Universal Robots PolyScope program: TEST_SUB_106B.urp

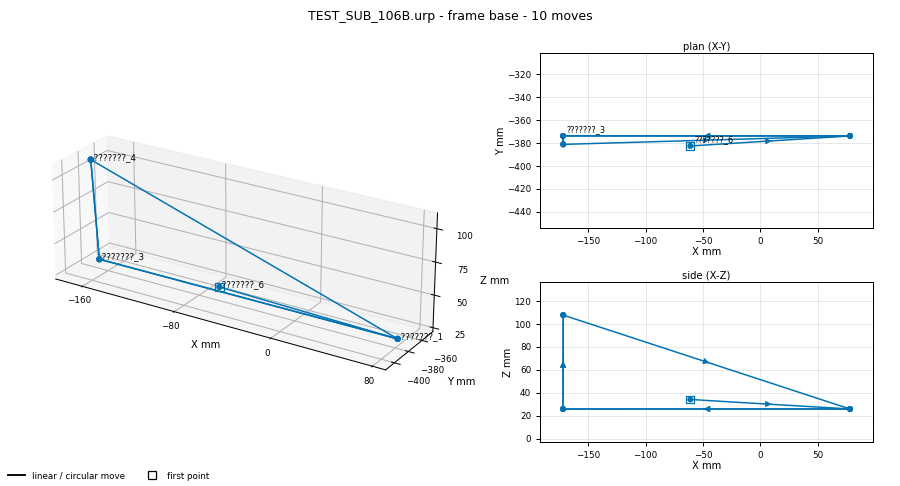
[picture p0: tool path of TEST_SUB_106B.urp in frame base, 10 of 10 moves have a stored position in this frame; points joined in program order, loops and branches not executed]
Program TEST_SUB_106B (installation=GD directory=/programs/GD createdIn=5.13.0 lastSavedIn=5.13.0 robotSerialNumber=20205000017)
Calibrated DH parameters: a=[-0.000157, -0.56303, -0.236706, -0.000074, -0.000109, 0]; d=[0.181705, 47.632387, 369.599619, -417.058513, 0.119878, 0.115667]; alpha=[1.570881, -0.005074, -0.001247, 1.56886, -1.570997, 0]; deltaTheta=[0, -0.405485, 5.544791, 1.143886, -0.000009, -0.000001]
InitVariablesNode
BeforeStart
  Script file /home/ros/ursim-5.13.0.113898/programs/GD/CONTROL/ALIGN_AXIS.script
    | def GET_NORM_VEC(p,axis=2):
    |   rot=p[0.0, 0.0, 0.0, p[3], p[4], p[5]]
    |   vec=p[0.0, 0.0, 0.0, 0.0, 0.0, 0.0]
    |   vec[axis]=1.0
    |   norm_p=pose_trans(rot,vec)
    |   return [norm_p[0], norm_p[1], norm_p[2]]
    | end
    | 
    | def GET_INNER_PRODUCT(v1,v2):
    |   return v1[0]*v2[0]+v1[1]*v2[1]+v1[2]*v2[2]
    | end
    | def GET_OUTER_PRODUCT(v1,v2):
    |   x=v1[1]*v2[2]-v1[2]*v2[1]
    |   y=v1[2]*v2[0]-v1[0]*v2[2]
    |   z=v1[0]*v2[1]-v1[1]*v2[0]
    |   return [x,y,z]
    | end
    | def GET_THETA(v1,v2):
    | #  cos=GET_INNER_PRODUCT(v1,v2) / norm(v1) / norm(v2)
    |   cos=GET_INNER_PRODUCT(v1,v2)
    |   g_cos=cos
    |   theta=norm(acos(cos))
    |   return theta
    | end
    | 
    | def GET_ALIGNED_POSE(target,feature,axis=2):
    |   feature_from_target=pose_trans(pose_inv(target),feature)
    |   g_f_from_t=feature_from_target
    |   nz_feature_from_target=GET_NORM_VEC(feature_from_target,axis)
    |   g_nz_f_from_t=nz_feature_from_target
    |   nz_target_from_target=[0.0, 0.0, 0.0]
    |   nz_target_from_target[axis]=1.0
    |   g_nz_t_from_t=nz_target_from_target
    | 
    |   theta=GET_THETA(nz_feature_from_target,nz_target_from_target)
    |   g_theta=theta
    |   rot_vec_n=normalize(GET_OUTER_PRODUCT(nz_target_from_target,nz_feature_from_target))
    | 
    |   if theta>d2r(90.0):
    |     theta=theta-d2r(180.0)
    |   end
    |   rot_vec=rot_vec_n * (theta)
    |   rot_p=p[0.0,0.0,0.0,rot_vec[0],rot_vec[1],rot_vec[2]]
    |   return pose_trans(target,rot_p)
    | end
    | def GET_ALIGNED_TCP(feature,axis=2):
    |   tcp=get_actual_tcp_pose()
    |   return GET_ALIGNED_POSE(tcp,feature,axis)
    | end
  Script file /home/ros/ursim-5.13.0.113898/programs/GD/CONTROL/align_axis_2.script
    | def get_normal_vector(pose, axis=2):
    |  rot = p[0.0, 0.0, 0.0, pose[3], pose[4], pose[5]]
    | 
    |  v = p[0.0, 0.0, 0.0, 0.0, 0.0, 0.0]
    |  if axis==0:
    |   v[0] = 1.0
    |  elif axis==1:
    |   v[1] = 1.0
    |  else:
    |   v[2] = 1.0
    |  end
    | 
    |  normal_p = pose_trans(rot, v)
    |  normal_vector = [normal_p[0], normal_p[1], normal_p[2]]
    |  return normal_vector
    | end
    | 
    | def get_inner_product(v1, v2):
    |  return v1[0]*v2[0] + v1[1]*v2[1] + v1[2]*v2[2]
    | end
    | 
    | def get_theta(v1, v2):
    |  cos = get_inner_product(v1, v2) / norm(v1) / norm(v2)
    |  theta_pn = acos(cos)
    |  theta = norm(theta_pn)
    |  return theta
    | end
    | 
    | def get_outer_product(v1, v2):
    |  x = v1[1]*v2[2] - v1[2]*v2[1]
    |  y = v1[2]*v2[0] - v1[0]*v2[2]
    |  z = v1[0]*v2[1] - v1[1]*v2[0]
    |  return [x,y,z]
    | end
    | 
    | def get_aligned_pose_current_to_base(axis=2):
    |  base = p[0.0, 0.0, 0.0, 0.0, 0.0, 0.0]
    |  pose_cur = get_actual_tcp_pose()
    |  return get_aligned_pose_to_axis(pose_cur, base, axis)
    | end
    | 
    | def get_aligned_pose_current_to_ref(pose_ref, axis=2):
    |  pose_cur = get_actual_tcp_pose()
    |  return get_aligned_pose_to_axis(pose_cur, pose_ref, axis)
    | end
    | 
    | def get_aligned_pose_to_axis(pose_target, pose_ref, axis=2):
    |  pose_ref_from_target = pose_trans(pose_inv(pose_target), pose_ref)
    |  nz_ref_from_target =  get_normal_vector(pose_ref_from_target, axis)
    |  nz_target_from_target = [0.0, 0.0, 1.0]
    | 
    |  if axis == 0:
    |   nz_target_from_target = [1.0, 0.0, 0.0]
    |  elif axis == 1:
    |   nz_target_from_target = [0.0, 1.0, 0.0]
    |  end
    | 
    |  theta = get_theta(nz_ref_from_target, nz_target_from_target)
    |  rot_vector_n = normalize(get_outer_product(nz_target_from_target, nz_ref_from_target))
    | 
    |  if theta > d2r(90.0):
    |   theta = theta - d2r(180.0)
    |  end
    | 
    |  rot_vector = rot_vector_n * (theta)
    | 
    |  pose_rot = p[0.0, 0.0, 0.0, rot_vector[0], rot_vector[1], rot_vector[2]]
    | 
    |  pose_aligned = pose_trans(pose_target, pose_rot)
    | 
    |  return pose_aligned
    | 
    | end
Robot Program (runOnlyOnce=false)
  MoveL speed 250 mm/s, acceleration 50 mm/s^2 (useActiveTCP=false) tcp=TCP_1; feature=Base
    SuppressedNode
      Waypoint ウェイポイント_2: TCP in base x=-24.264 y=-372.872 z=25.863 mm, rx=-0.0592 ry=3.141 rz=-0.0002 rad; joints [-70.474, -66.693, -131.957, -71.332, 89.989, 17.477] deg; TCP offset x=0 y=80 z=420 mm, rx=0 ry=0 rz=0 rad
    SuppressedNode
      Wait Sleep waitTime=0.5
    Waypoint ウェイポイント_6: TCP in base x=-61.068 y=-382.464 z=34.138 mm, rx=0.7542 ry=-2.9409 rz=0.2397 rad; joints [-59.813, -53.273, -138.338, -71.164, 82.262, 0.931] deg
    Wait Sleep waitTime=0.5
  var_5 := p[0.0,0.0,0.0,0.0,0.0,0.0]
  SuppressedNode
    Script: var_5=get_actual_tool_flange_pose()
  SuppressedNode
    Script: var_5[0]=0
  SuppressedNode
    Script: var_5[1]=0
  SuppressedNode
    Script: var_5[0]=0
  Wait Sleep waitTime=0.5
  Set NoAction tcp=TCP_1
  var_4 := GET_ALIGNED_TCP(var_5)
  Wait Sleep waitTime=5
  var_20 := pose_sub(CurrPos,var_4)
  var_21 := pose_trans(pose_inv(CurrPos),var_4)
  Set NoAction tcp=ZERO
  var_1 := get_tcp_offset()
  var_7 := pose_trans(var_1, var_21)
  SuppressedNode
    var_7 := get_aligned_pose_current_to_base()
  SuppressedNode
    MoveL speed 250 mm/s, acceleration 50 mm/s^2 (useActiveTCP=true) feature=Base
      SuppressedNode
        Waypoint ウェイポイント_2: TCP in base x=-24.264 y=-372.872 z=25.863 mm, rx=-0.0592 ry=3.141 rz=-0.0002 rad; joints [-70.474, -66.693, -131.957, -71.332, 89.989, 17.477] deg
      SuppressedNode
        Wait Sleep waitTime=0.5
      Waypoint ウェイポイント_6: TCP in base x=0.269 y=-378.011 z=457.243 mm, rx=0.7542 ry=-2.9409 rz=0.2397 rad; joints [-59.813, -53.273, -138.338, -71.164, 82.262, 0.931] deg
      Wait Sleep waitTime=2
      SuppressedNode
        Waypoint Variable (Variable): variable=var_4
      SuppressedNode
        Wait Sleep waitTime=0.5
  MoveL speed 250 mm/s, acceleration 50 mm/s^2 (useActiveTCP=false) tcp=TCP_1; feature=Base
    Waypoint ウェイポイント_1: TCP in base x=78.379 y=-373.699 z=25.825 mm, rx=-0.2371 ry=3.1325 rz=-0.0004 rad; joints [-56.545, -67.63, -131.248, -71.107, 89.997, 24.798] deg; TCP offset x=0 y=80 z=420 mm, rx=0 ry=0 rz=0 rad
    SuppressedNode
      p1 := CurrPos_p
    Wait Sleep waitTime=1
    SuppressedNode
      p11 := GET_ALIGNED_TCP(p1)
  Script: set_tcp(var_7)
  MoveL speed 250 mm/s, acceleration 50 mm/s^2 (useActiveTCP=true) feature=Base
    Waypoint ウェイポイント_1: TCP in base x=78.379 y=-373.699 z=25.825 mm, rx=-0.2371 ry=3.1325 rz=-0.0004 rad; joints [-56.545, -67.63, -131.248, -71.107, 89.997, 24.798] deg
    Wait Sleep waitTime=1
    SuppressedNode
      Waypoint Variable (Variable): variable=p1
    SuppressedNode
      Wait Sleep waitTime=1
    SuppressedNode
      Waypoint Variable (Variable): variable(name=p11)
    SuppressedNode
      Wait Sleep waitTime=1
    Popup Message (haltProgram=false message=1 done inputType=Text)
  Set NoAction tcp=ZERO
  MoveL speed 250 mm/s, acceleration 50 mm/s^2 (useActiveTCP=false) tcp=TCP_1; feature=Base
    Waypoint ウェイポイント_3: TCP in base x=-172.242 y=-373.664 z=25.794 mm, rx=-0.2375 ry=3.1326 rz=-0.0004 rad; joints [-88.225, -69.95, -129.885, -70.151, 90.002, -6.895] deg
    SuppressedNode
      p2 := CurrPos_p
    Wait Sleep waitTime=1
    SuppressedNode
      p12 := GET_ALIGNED_TCP(p2)
  Script: set_tcp(var_7)
  MoveL speed 250 mm/s, acceleration 50 mm/s^2 (useActiveTCP=true) feature=Base
    Waypoint ウェイポイント_3: TCP in base x=-172.242 y=-373.664 z=25.794 mm, rx=-0.2375 ry=3.1326 rz=-0.0004 rad; joints [-88.225, -69.95, -129.885, -70.151, 90.002, -6.895] deg
    Wait Sleep waitTime=1
    SuppressedNode
      Waypoint Variable (Variable): variable=p2
    SuppressedNode
      Wait Sleep waitTime=1
    SuppressedNode
      Waypoint Variable (Variable): variable(name=p12)
    SuppressedNode
      Wait Sleep waitTime=1
    Popup Message (haltProgram=false message=2 done inputType=Text)
  Set NoAction tcp=ZERO
  MoveL speed 250 mm/s, acceleration 50 mm/s^2 (useActiveTCP=false) tcp=TCP_1; feature=Base
    Waypoint ウェイポイント_4: TCP in base x=-172.007 y=-381.075 z=107.802 mm, rx=-0.2377 ry=3.1326 rz=-0.0003 rad; joints [-88.222, -68.286, -122.359, -79.345, 90.002, -6.902] deg
    SuppressedNode
      p3 := CurrPos_p
    Wait Sleep waitTime=1
    SuppressedNode
      p13 := GET_ALIGNED_TCP(p3)
  Script: set_tcp(var_7)
  MoveL speed 250 mm/s, acceleration 50 mm/s^2 (useActiveTCP=true) feature=Base
    Waypoint ウェイポイント_4: TCP in base x=-172.007 y=-381.075 z=107.802 mm, rx=-0.2377 ry=3.1326 rz=-0.0003 rad; joints [-88.222, -68.286, -122.359, -79.345, 90.002, -6.902] deg
    Wait Sleep waitTime=1
    SuppressedNode
      Waypoint Variable (Variable): variable=p3
    SuppressedNode
      Wait Sleep waitTime=1
    SuppressedNode
      Waypoint Variable (Variable): variable(name=p13)
    SuppressedNode
      Wait Sleep waitTime=1
    Popup Message (haltProgram=false message=3 done inputType=Text)
  Script: CurrPos=get_actual_tool_flange_pose()
  CutOffPos := CurrPos
  var_1 := get_tcp_offset()
  var_2 := pose_trans(CutOffPos,var_1)
  SuppressedNode
    Folder FREE_DRIVE
      Script: freedrive_mode()
      SetPayload (workpieceName=k2)
      Set NoAction tcp=ZERO
      Wait Sleep waitTime=1
      Script: end_freedrive_mode()
      Wait Condition expression=is_steady()
  SetPayload (workpieceName=k10)
  Set NoAction tcp=TCP_1
  Wait Sleep waitTime=0.5
  Folder CUTOFF_POSE
    CutOffPos := CurrPos
    var_6 := CutOffPos
    SuppressedNode
      CutOffPos := p[0.0,0.0,0.0,CutOffPos[3],CutOffPos[4],CutOffPos[5]]
    var_1 := get_tcp_offset()
    var_20 := pose_trans(pose_inv(CutOffPos),var_1)
    SuppressedNode
      CutOffPos := 
    var_4 := p[0.0,0.0,0.0,CutOffPos[3],CutOffPos[4],CutOffPos[5]]
    var_5 := p[0.0,0.0,0.0,0.0,0.0,CutOffPos[5]]
    CutOffPos := pose_trans(var_4,pose_inv(var_5))
    SuppressedNode
      CutOffPos := p[0.0,0.0,0.0,var_5[0],var_5[1],var_5[2]]
    var_20 := pose_trans(pose_inv(CutOffPos),var_1)
    var_21 := pose_trans(var_1,CutOffPos)
    var_2 := pose_trans(CutOffPos,var_1)
  Wait Condition expression=is_steady()
  SuppressedNode
    Script: CurrPos_p=get_actual_tcp_pose()
  SuppressedNode
    CircleMove (OrientationMode=UNCONSTRAINED)
  Script: set_tcp(var_2)
  SuppressedNode
    Folder TRANSFER
      Timer (action=Reset) variable(name=tm_relmove)
      Timer (action=Start) variable=tm_relmove
      ForceStartZ := CurrPos_p[2]
      Force Frame feature=Bucket; selection=[0, 0, 1, 0, 0, 0]; wrench=[0, 0, 40, 0, 0, 0]; limitsForce=[0.01, 0.01, 0.25, 0.174533, 0.174533, 0.174533]; limitsMotion=[0.1, 0.1, 0.1, 0.349066, 0.349066, 0.349066]
        Wait Condition expression=tm_relmove>GPII_TMCutOff or CurrPos_p[2]>ForceStartZ+RelMoveZ
      Timer (action=Stop) variable=tm_relmove
      If (WorkPosNo≟0)
        MoveL speed 60 mm/s, acceleration 15 mm/s^2 (useActiveTCP=false) tcp=ZERO; feature=Base
          PoseSub := pose_sub(CurrPos, pose_trans(g2GD_pos5, pose_inv(get_tcp_offset())))
          RZSub := r2d(PoseSub[5])
          If (norm(PoseSub[5])≥d2r(RZTh))
            Script: PoseSub[0]=0.0
            Script: PoseSub[1]=0.0
            Script: PoseSub[2]=0.0
            PoseAdd := pose_add(PoseSub, CurrPos)
            Waypoint Variable (Variable): variable=PoseAdd
        MoveL speed 250 mm/s, acceleration 50 mm/s^2 (useActiveTCP=false) tcp=TCP_1; feature=Base
          Waypoint Variable (Variable): variable(featureName=g2GD_pos5)
        MoveL speed 400 mm/s, acceleration 140 mm/s^2 (useActiveTCP=false) tcp=TCP_1; feature=Base
          SetPayload (workpieceName=k10)
          Waypoint Variable (Variable): variable(featureName=g2GD_pos4)
          Waypoint Variable (Variable): motionParameters(blendRadius=0.1); variable(featureName=g2GD_pos3)
          Waypoint Variable (Variable): motionParameters(jointSpeed=1.047198 jointAcceleration=1.396263 cartesianSpeed=0.4 cartesianAcceleration=0.07); variable(featureName=g2GD_pos2)
        MoveL speed 400 mm/s, acceleration 70 mm/s^2 (useActiveTCP=false) tcp=TCP_1; feature=Base
          SetPayload (workpieceName=k120)
          Waypoint Variable (Variable): motionParameters(blendRadius=0.05); variable(featureName=g2GD_pos1)
      ElseIf (WorkPosNo≟1)
        MoveL speed 60 mm/s, acceleration 15 mm/s^2 (useActiveTCP=false) tcp=ZERO; feature=Base
          PoseSub := pose_sub(CurrPos, pose_trans(g1GD_pos5, pose_inv(get_tcp_offset())))
          RZSub := r2d(PoseSub[5])
          If (norm(PoseSub[5])≥d2r(RZTh))
            Script: PoseSub[0]=0.0
            Script: PoseSub[1]=0.0
            Script: PoseSub[2]=0.0
            PoseAdd := pose_add(PoseSub, CurrPos)
            Waypoint Variable (Variable): variable=PoseAdd
        MoveL speed 250 mm/s, acceleration 50 mm/s^2 (useActiveTCP=false) tcp=TCP_1; feature=Base
          Waypoint Variable (Variable): variable(featureName=g1GD_pos5)
        MoveL speed 400 mm/s, acceleration 140 mm/s^2 (useActiveTCP=false) tcp=TCP_1; feature=Base
          SetPayload (workpieceName=k10)
          Waypoint Variable (Variable): variable(featureName=g1GD_pos3)
          Waypoint Variable (Variable): variable(featureName=g1GD_pos2)
        MoveL speed 400 mm/s, acceleration 140 mm/s^2 (useActiveTCP=false) tcp=TCP_1; feature=Base
          SetPayload (workpieceName=k120)
          Waypoint Variable (Variable): motionParameters(blendRadius=0.1); variable(featureName=g1GD_pos1)
  MoveL speed 250 mm/s, acceleration 50 mm/s^2 (useActiveTCP=true) feature=Base
    var_3 := get_tcp_offset()
    Waypoint ウェイポイント_1: TCP in base x=78.379 y=-373.699 z=25.825 mm, rx=-0.2371 ry=3.1325 rz=-0.0004 rad; joints [-56.545, -67.63, -131.248, -71.107, 89.997, 24.798] deg
    Wait Sleep waitTime=1
    Waypoint ウェイポイント_3: TCP in base x=-172.242 y=-373.664 z=25.794 mm, rx=-0.2375 ry=3.1326 rz=-0.0004 rad; joints [-88.225, -69.95, -129.885, -70.151, 90.002, -6.895] deg
    Wait Sleep waitTime=1
    Waypoint ウェイポイント_4: TCP in base x=-172.007 y=-381.075 z=107.802 mm, rx=-0.2377 ry=3.1326 rz=-0.0003 rad; joints [-88.222, -68.286, -122.359, -79.345, 90.002, -6.902] deg
    Wait Sleep waitTime=1
  Popup Message (haltProgram=false message=done! inputType=Text)
Thread スレッド_1 (runOnlyOnce=false)
  Script: CurrPos=get_actual_tool_flange_pose()
  Script: CurrPos_p=get_actual_tcp_pose()
  Script: sync()
